ABB RobotStudio station: themal simulation.rspag

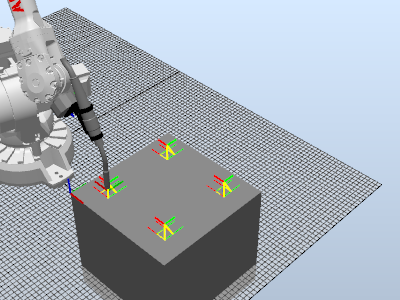
--- station ---
Station themal simulation (saved by RobotStudio 22.2.9947.0)
Controller IRB2600_12_185
  mechanical unit ROB_1: IRB2600_12_185__02, 6 joints, base frame (0, 0, 0) mm
Layout (positions relative to the parent item):
  - IRB2600_12_185__02 [mechanism, from Robots\IRB2600_12_185_G_02.rslib] at (0, 0, 0) mm; joint values [-0.2959, -0.2098, 1.1048, 2.3622, 0.3432, -2.5687] (rad or m)
  - AW_Gun_PSF_25 [mechanism, from Tools\AW_Gun_PSF_25.rslib] at (594.64, -160.23, 727.24) mm, rotated rx 180 ry 54.2 rz 180 deg
  - Part_1 [part] at (100, 0, -100) mm, size 500 x 500 x 500 mm
Attachment: AW_Gun_PSF_25 is attached to IRB2600_12_185__02 / Link6

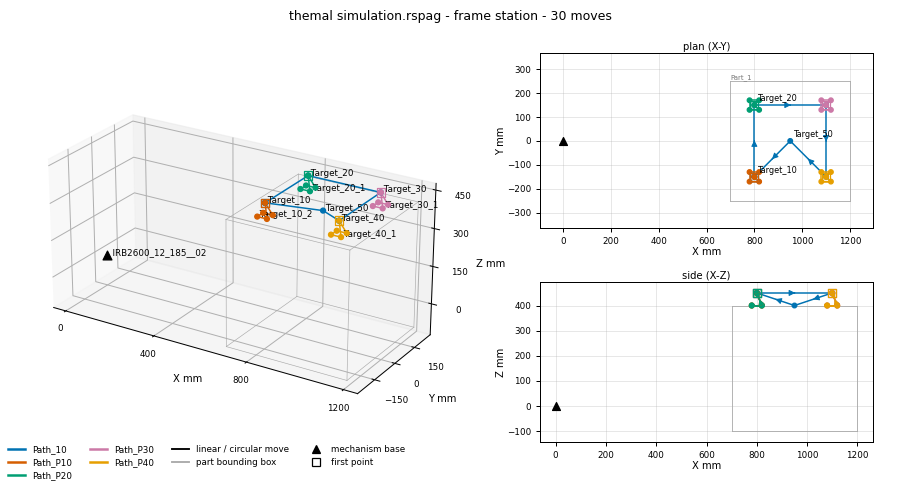
[picture p0: tool path of themal simulation.rspag in frame station, 30 of 30 moves have a stored position in this frame; points joined in program order, loops and branches not executed]
--- Controller Data/IRB2600_12_185/RAPID/TASK1/PROGMOD/CalibData.mod ---
MODULE CalibData
    PERS tooldata AW_Gun:=[TRUE,[[119.5,0,352],[0.890213743,0,0.455543074,0]],[1,[0,0,100],[1,0,0,0],0,0,0]];
    TASK PERS wobjdata wobjWelding:=[FALSE,TRUE,"",[[700,-250,400],[1,0,0,0]],[[0,0,0],[1,0,0,0]]];
ENDMODULE

--- Controller Data/IRB2600_12_185/RAPID/TASK1/PROGMOD/Module1.mod ---
MODULE Module1
        CONST robtarget Target_10:=[[100,100,50],[0,0,1,0],[-1,1,-2,0],[9E+09,9E+09,9E+09,9E+09,9E+09,9E+09]];
    CONST robtarget Target_20:=[[100,400,50],[0,0,1,0],[0,2,-3,0],[9E+09,9E+09,9E+09,9E+09,9E+09,9E+09]];
    CONST robtarget Target_30:=[[400,400,50],[0,0,1,0],[0,2,-3,0],[9E+09,9E+09,9E+09,9E+09,9E+09,9E+09]];
    CONST robtarget Target_40:=[[400,100,50],[0,0,1,0],[-1,1,-2,0],[9E+09,9E+09,9E+09,9E+09,9E+09,9E+09]];
    CONST robtarget Target_50:=[[250,250,0],[0,0,1,0],[0,1,-2,0],[9E+09,9E+09,9E+09,9E+09,9E+09,9E+09]];
    CONST robtarget Target_10_1:=[[120,80,0],[0,0,1,0],[-1,1,-2,0],[9E+09,9E+09,9E+09,9E+09,9E+09,9E+09]];
    CONST robtarget Target_10_2:=[[80,80,0],[0,0,1,0],[-1,1,-2,0],[9E+09,9E+09,9E+09,9E+09,9E+09,9E+09]];
    CONST robtarget Target_10_3:=[[80,120,0],[0,0,1,0],[-1,1,-2,0],[9E+09,9E+09,9E+09,9E+09,9E+09,9E+09]];
    CONST robtarget Target_10_4:=[[120,120,0],[0,0,1,0],[-1,1,-2,0],[9E+09,9E+09,9E+09,9E+09,9E+09,9E+09]];
    CONST robtarget Target_20_1:=[[120,380,0],[0,0,1,0],[0,2,-3,0],[9E+09,9E+09,9E+09,9E+09,9E+09,9E+09]];
    CONST robtarget Target_20_2:=[[80,380,0],[0,0,1,0],[0,2,-3,0],[9E+09,9E+09,9E+09,9E+09,9E+09,9E+09]];
    CONST robtarget Target_20_3:=[[80,420,0],[0,0,1,0],[0,2,-3,0],[9E+09,9E+09,9E+09,9E+09,9E+09,9E+09]];
    CONST robtarget Target_20_4:=[[120,420,0],[0,0,1,0],[0,2,-3,0],[9E+09,9E+09,9E+09,9E+09,9E+09,9E+09]];
    CONST robtarget Target_30_1:=[[420,380,0],[0,0,1,0],[0,2,-3,0],[9E+09,9E+09,9E+09,9E+09,9E+09,9E+09]];
    CONST robtarget Target_30_2:=[[380,380,0],[0,0,1,0],[0,2,-3,0],[9E+09,9E+09,9E+09,9E+09,9E+09,9E+09]];
    CONST robtarget Target_30_3:=[[380,420,0],[0,0,1,0],[0,2,-3,0],[9E+09,9E+09,9E+09,9E+09,9E+09,9E+09]];
    CONST robtarget Target_30_4:=[[420,420,0],[0,0,1,0],[0,2,-3,0],[9E+09,9E+09,9E+09,9E+09,9E+09,9E+09]];
    CONST robtarget Target_40_1:=[[420,80,0],[0,0,1,0],[-1,1,-2,0],[9E+09,9E+09,9E+09,9E+09,9E+09,9E+09]];
    CONST robtarget Target_40_2:=[[380,80,0],[0,0,1,0],[-1,1,-2,0],[9E+09,9E+09,9E+09,9E+09,9E+09,9E+09]];
    CONST robtarget Target_40_3:=[[380,120,0],[0,0,1,0],[-1,1,-2,0],[9E+09,9E+09,9E+09,9E+09,9E+09,9E+09]];
    CONST robtarget Target_40_4:=[[420,120,0],[0,0,1,0],[-1,1,-2,0],[9E+09,9E+09,9E+09,9E+09,9E+09,9E+09]];
!***********************************************************
    !
    ! Module:  Module1
    !
    ! Description:
    !   <Insert description here>
    !
    ! Author: xizh0002
    !
    ! Version: 1.0
    !
    !***********************************************************


    !***********************************************************
    !
    ! Procedure main
    !
    !   This is the entry point of your program
    !
    !***********************************************************
    PROC main()
        FOR i FROM 1 TO 10 DO
            Path_P10;
        ENDFOR
        FOR i FROM 1 TO 10 DO
            Path_P20;
        ENDFOR
        FOR i FROM 1 TO 10 DO
            Path_P30;
        ENDFOR
        FOR i FROM 1 TO 10 DO
            Path_P40;
        ENDFOR
    ENDPROC
    PROC Path_10()
        MoveJ Target_10,v100,z10,AW_Gun\WObj:=wobjWelding;
        MoveL Target_20,v100,fine,AW_Gun\WObj:=wobjWelding;
        MoveL Target_30,v100,fine,AW_Gun\WObj:=wobjWelding;
        MoveL Target_40,v100,fine,AW_Gun\WObj:=wobjWelding;
        MoveL Target_50,v100,fine,AW_Gun\WObj:=wobjWelding;
        MoveL Target_10,v100,z10,AW_Gun\WObj:=wobjWelding;
    ENDPROC
    PROC Path_P10()
        MoveJ Target_10,v100,z10,AW_Gun\WObj:=wobjWelding;
        MoveL Target_10_1,v100,fine,AW_Gun\WObj:=wobjWelding;
        MoveL Target_10_2,v100,fine,AW_Gun\WObj:=wobjWelding;
        MoveL Target_10_3,v100,fine,AW_Gun\WObj:=wobjWelding;
        MoveL Target_10_4,v100,fine,AW_Gun\WObj:=wobjWelding;
        MoveL Target_10,v100,z10,AW_Gun\WObj:=wobjWelding;
    ENDPROC
    PROC Path_P20()
        MoveJ Target_20,v100,z10,AW_Gun\WObj:=wobjWelding;
        MoveL Target_20_1,v100,fine,AW_Gun\WObj:=wobjWelding;
        MoveL Target_20_2,v100,fine,AW_Gun\WObj:=wobjWelding;
        MoveL Target_20_3,v100,fine,AW_Gun\WObj:=wobjWelding;
        MoveL Target_20_4,v100,fine,AW_Gun\WObj:=wobjWelding;
        MoveL Target_20,v100,z10,AW_Gun\WObj:=wobjWelding;
    ENDPROC
    PROC Path_P30()
        MoveJ Target_30,v100,z10,AW_Gun\WObj:=wobjWelding;
        MoveL Target_30_1,v100,fine,AW_Gun\WObj:=wobjWelding;
        MoveL Target_30_2,v100,fine,AW_Gun\WObj:=wobjWelding;
        MoveL Target_30_3,v100,fine,AW_Gun\WObj:=wobjWelding;
        MoveL Target_30_4,v100,fine,AW_Gun\WObj:=wobjWelding;
        MoveL Target_30,v100,z10,AW_Gun\WObj:=wobjWelding;

    ENDPROC
    PROC Path_P40()
        MoveJ Target_40,v100,fine,AW_Gun\WObj:=wobjWelding;
        MoveL Target_40_1,v100,fine,AW_Gun\WObj:=wobjWelding;
        MoveL Target_40_2,v100,fine,AW_Gun\WObj:=wobjWelding;
        MoveL Target_40_3,v100,fine,AW_Gun\WObj:=wobjWelding;
        MoveL Target_40_4,v100,fine,AW_Gun\WObj:=wobjWelding;
        MoveL Target_40,v100,fine,AW_Gun\WObj:=wobjWelding;
    ENDPROC
ENDMODULE
